FUNCTION_BLOCK AOI_SensorAdmin
VAR_INPUT
END_VAR
VAR_OUTPUT
END_VAR
VAR
	TON_Fliter: TON;

END_VAR
VAR_IN_OUT
	Admin: UDT_SensorAdmin;
END_VAR

TON_Fliter(IN:= admin.i.Link, PT:=DINT_TO_TIME(admin.i.FilterTime) , Q=>admin.o.Value , ET=> );

END_FUNCTION_BLOCK

(* stored: Version 1.1.0.1, ProductVersion 3.1.4022.16
   POU AOI_SensorAdmin: Id {fd193fc9-d0b1-49fa-8a87-c9f0b51061eb}, SpecialFunc None *)
